// SIMATIC S7-200 project (STEP 7-Micro/WIN), CPU 226 REL 02.01

SYMBOL_TABLE USR1
Motor_START      I1.0     // The START button is attached to this input.
Motor_STOP       I1.1     // The STOP button is attached to this input.
Direction        I1.5     // If set, the motor runs counterclockwise. If not set, the motor runs clockwise.
Drive_ON         M0.1     // When memory bit M0.1 is set, the motor is turned on.
Blocking         M0.2     // This flag is set when Motor STOP is pressed. It turns the drive off immediately
Always_On        SM0.0    // This bit is always on.
First_Scan_On    SM0.1    // This bit is on for the first scan cycle only.
PLS0_Ctrl        SMB67    // Controls pulse train output & pulse width modulation functions for output Q0.0.
PLS0_Cycle       SMW68    // Cycle time value, pulse train or pls. width modulation output 0. SMB68 is MSB.
PWM0_PW          SMW70    // Pulse width value of pulse width modulation output 0. SMB70 is the MSB.
PTO0_PC          SMD72    // Pulse count value of pulse train output 0. SMB72 is the most significant byte.
END_SYMBOL_TABLE

ORGANIZATION_BLOCK MAIN:OB1
TITLE= Tip022B
//  题目：用集成脉冲输出触发步进电机驱动器
// ***概述***
//  CPU214有两个脉冲输出，可以用来产生控制步进电机驱动器的脉冲。功率驱
// 动器将控制脉冲按照某种模式转换成步进电机线圈的电流，产生旋转磁场，使得
// 转子只能按固定的步数(步数a)来改变它的位置。连续的脉冲序列产生与其对应
// 的同频率（同步机）步序列。如果控制频率足够高，步进电机的转动可看作一个
// 连续的转动。
// 本例叙述用Q0.0的输出脉冲触发步进电机驱动器。当输入端I1.0发出"START"信号后，
// 控制器将输出固定数目的方波脉冲，使步进电机按对应的步数转动。当输入端I1.1
// 发出“STOP”信号后，步进电机停止转动。接在输入端I1.5的方向开关位置决定电机
// 正转或反转。
// 硬件要求
// 数量               设备               制造厂/订货号
//  1          SIMATIC S7-200 CPU-214     SIEMENS/6ES7 214-1AC00-0XB0
//  1          PC/PPI电缆                 SIEMENS/6ES7 901-3BF00-0XA0
//  1          编程设备或PC 
//  1          带有标准的功率驱动器和相关连接电缆的步进电机
//  1          用于传输控制信号到功率驱动器的电缆
//  1          开关
//  2          按钮
// 
// ***程序和注释***
//  1. 初始化  
//   在程序的第一个扫描周期(SM0.1=1),为两种脉冲输出功能（PTO和PTW）选择参
// 数，本例从中选择了PTO, 并规定了脉冲周期和脉冲数。
//  2. 选择旋转方向
//   用接在输入端I1.5的开关来选择转动方向。如果I1.5=1,将输出Q0.2置成高电位
// 那么电机逆时针转动。如果I1.5=0,将输出Q0.2置成低电位，那么电机顺时针转动。
// 为保护电机避免漏步，电机转动方向的改变只能在电机处于停止状态(M0.1=0)时
// 进行。
//  3. 起动电机
//  起动电机的三个条件如下：
//         (1) 按"START"(起动)按钮，在输入端I1.0产生脉冲上升沿(从0升到1);
//         (2) 无联锁，即联锁标志M0.2=0;
//         (3) 电机处于停止状态，即操作标志M0.1=0。
//  如果同时具备上述3个条件，则将M0.1置位(M0.1=1),控制器执行PLS0指令，在输出端
// Q0.0输出脉冲，其他必须预先具备的条件，已经在首次扫描(SM0.1=1)设置，主要是脉
// 冲输出功能的基本数据。例如，时基、周期和脉冲数。这些数据置于相应的属于PTO/PWM的
// 特殊存储字SMW68,SMW70和SMD72。
// 4. 停止电机
//  停止电机的两个条件如下：
//      (1)  按"STOP"按钮，在输入端I1.1产生脉冲上升沿(从0升到1);
//      (2)  电机处于运转状态，即操作标志M0.1=1。
// 如果同时具备上述2个条件，则将标志M0.1复位(M0.1=0),并中断输出端Q0.0的脉冲输出。
// 这与执行PLS0命令有关，它将脉宽调制(PWM)输出的脉冲宽度减为0(所需的基本设置已在第
// 一扫描周期中定义了),因而输出信号被抑制。
//  在完整的脉冲序列输出后，中断程序0将标志M0.1复位(M0.1=0),从而使电机能够重新起动。
//  5.联锁
//  为保护人员和设备的安全，再按"STOP"(停止)按钮(I1.1)之后，必须规定驱动器连锁(或称
// 阻塞),将联锁标志M0.2置位(M0.2=1),立即关断驱动器。只有在M0.2复位，(M0.2=0)后，才能
// 重新起动电机。当"STOP"按钮松开后，为防止电机的意外起动，只有在“START”(I1.0)和
// "STOP"按钮(I1.1)都松开后，才能将M0.2复位(M0.2=0),如果要再次起动电机，则必须再发出
// 一个起动信号。
//  6.程序清单
// 本程序长度为64个字
// 标题：驱动器功能测试
// 
BEGIN
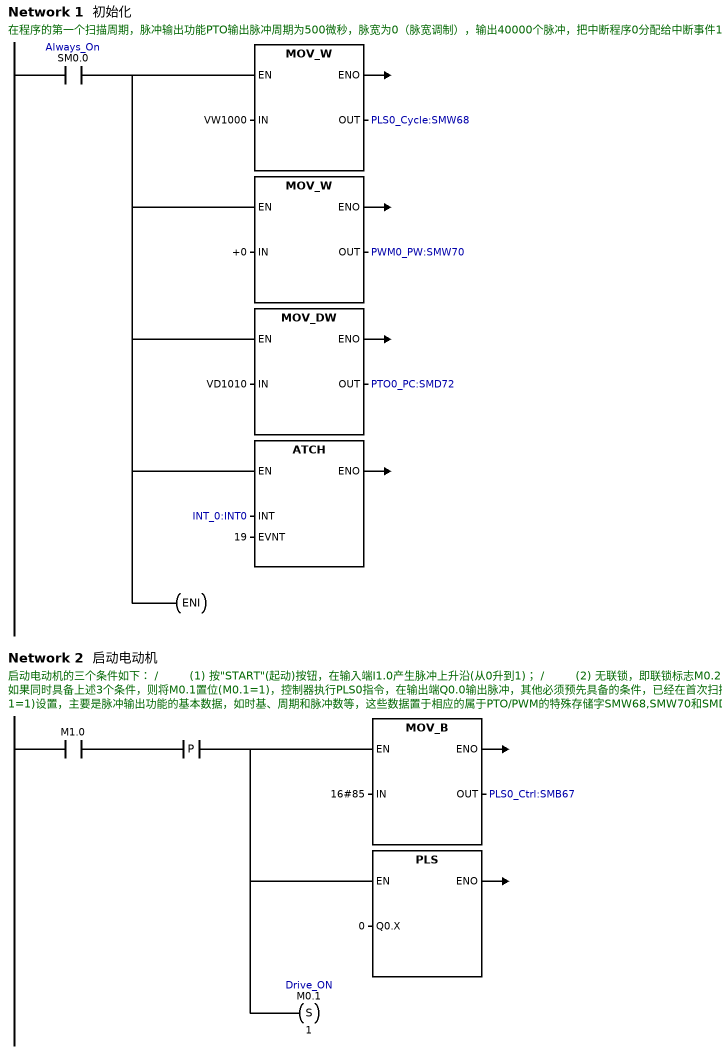
Network 1 // 初始化
// 在程序的第一个扫描周期，脉冲输出功能PTO输出脉冲周期为500微秒，脉宽为0（脉宽调制），输出40000个脉冲，把中断程序0分配给中断事件19（PLS0 脉冲输出结束），允许中断
// 仅首次扫描周期SM0.1置位(SM0.1=1)
// 输出脉冲周期为500微秒
// 脉宽为0（脉宽调制）
// 输出40000个脉冲
// 把中断程序0分配给中断事件19（PLS0
// 脉冲输出结束）
// 允许中断
LD     Always_On:SM0.0
MOVW   VW1000, PLS0_Cycle:SMW68
MOVW   +0, PWM0_PW:SMW70
MOVD   VD1010, PTO0_PC:SMD72
ATCH   INT_0:INT0, 19
ENI
Network 2 // 启动电动机
// 启动电动机的三个条件如下：
//         (1) 按"START"(起动)按钮，在输入端I1.0产生脉冲上升沿(从0升到1)；
//         (2) 无联锁，即联锁标志M0.2=0；
//         (3) 电机处于停止状态，即操作标志M0.1=0。
// 如果同时具备上述3个条件，则将M0.1置位(M0.1=1)，控制器执行PLS0指令，在输出端Q0.0输出脉冲，其他必须预先具备的条件，已经在首次扫描(SM0.1=1)设置，主要是脉冲输出功能的基本数据，如时基、周期和脉冲数等，这些数据置于相应的属于PTO/PWM的特殊存储字SMW68,SMW70和SMD72
// 若按"START"(起动)按钮
// 上升沿
// 且无联锁
// 且电机停止 则
// 置脉冲输出功能的控制位
// 起动脉冲输出(Q0.0)
// 电机运行标志M0.1置位(M0.1=1)
LD     M1.0
EU
MOVB   16#85, PLS0_Ctrl:SMB67
PLS    0
S      Drive_ON:M0.1, 1
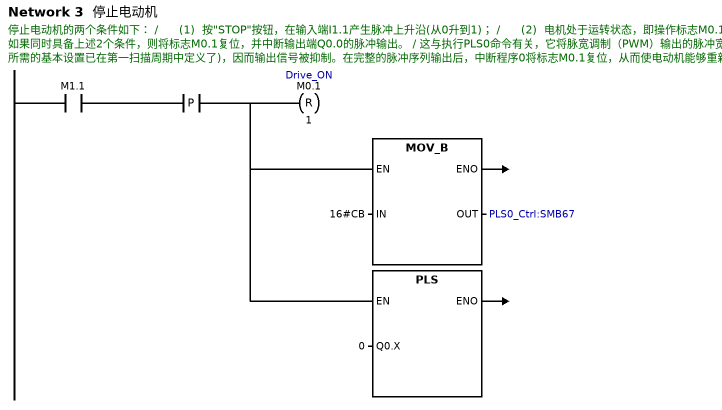
Network 3 // 停止电动机
//  停止电动机的两个条件如下：
//      (1)  按"STOP"按钮，在输入端I1.1产生脉冲上升沿(从0升到1)；
//      (2)  电机处于运转状态，即操作标志M0.1=1。
// 如果同时具备上述2个条件，则将标志M0.1复位，并中断输出端Q0.0的脉冲输出。
// 这与执行PLS0命令有关，它将脉宽调制（PWM）输出的脉冲宽度减为0(所需的基本设置已在第一扫描周期中定义了)，因而输出信号被抑制。在完整的脉冲序列输出后，中断程序0将标志M0.1复位，从而使电动机能够重新启动。
// 若按"STOP"(停止)按钮，
// 上升沿
// 且电机正在转动，则
// 电机运行标志M0.1复位(M0.1=0)
// 置脉冲输出功能的控制位，PWM的脉宽为0
// 输出端Q0.0无脉冲
LD     M1.1
EU
R      Drive_ON:M0.1, 1
MOVB   16#CB, PLS0_Ctrl:SMB67
PLS    0
Network 4 //  主程序结束
// MEND				
// 
Network 5 // ***中断程序0***
END_ORGANIZATION_BLOCK

INTERRUPT_BLOCK INT_0:INT0
TITLE=
BEGIN
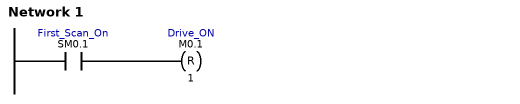
Network 1
// 电机运行标志M0.1复位(M0.1=0)
LD     First_Scan_On:SM0.1
R      Drive_ON:M0.1, 1
Network 2 //  中断程序0结束
// RETI					
// 
END_INTERRUPT_BLOCK
